{attribute addProperty BoxType "EP9224-0023-0016"}
{attribute addProperty Id "Temperature_WarningAT %I*BOOL811Temperature_ErrorAT %I*BOOL812Us_WarningAT %I*BOOL813Us_ErrorAT %I*BOOL814Up_WarningAT %I*BOOL815Up_ErrorAT %I*BOOL816Global_Error_BitAT %I*BOOL817Sum_Current_WarningAT %I*BOOL818Sum_Current_ErrorAT %I*BOOL819Reset_InputAT %I*BOOL8112TxPDO_StateAT %I*BOOL8115TxPDO_ToggleAT %I*BOOL8116Current_UsAT %I*INT16217Current_UpAT %I*INT16218Voltage_UsAT %I*INT16219Voltage_UpAT %I*INT16220TemperatureAT %I*INT16221"}
{attribute addProperty CRC "807253555"}
{attribute addProperty SizeInBites "176"}
{attribute addProperty SizeInBytes "22"}
TYPE DPO_Inputs_Device_301DB633 :
STRUCT
	{attribute addProperty Name "Temperature_Warning"}
	Temperature_Warning AT %I* : BOOL;
	{attribute addProperty Name "Temperature_Error"}
	Temperature_Error AT %I* : BOOL;
	{attribute addProperty Name "Us_Warning"}
	Us_Warning AT %I* : BOOL;
	{attribute addProperty Name "Us_Error"}
	Us_Error AT %I* : BOOL;
	{attribute addProperty Name "Up_Warning"}
	Up_Warning AT %I* : BOOL;
	{attribute addProperty Name "Up_Error"}
	Up_Error AT %I* : BOOL;
	{attribute addProperty Name "Global_Error_Bit"}
	Global_Error_Bit AT %I* : BOOL;
	{attribute addProperty Name "Sum_Current_Warning"}
	Sum_Current_Warning AT %I* : BOOL;
	{attribute addProperty Name "Sum_Current_Error"}
	Sum_Current_Error AT %I* : BOOL;
	{attribute addProperty Name "Reset_Input"}
	Reset_Input AT %I* : BOOL;
	{attribute addProperty Name "TxPDO_State"}
	TxPDO_State AT %I* : BOOL;
	{attribute addProperty Name "TxPDO_Toggle"}
	TxPDO_Toggle AT %I* : BOOL;
	{attribute addProperty Name "Current_Us"}
	Current_Us AT %I* : INT;
	{attribute addProperty Name "Current_Up"}
	Current_Up AT %I* : INT;
	{attribute addProperty Name "Voltage_Us"}
	Voltage_Us AT %I* : INT;
	{attribute addProperty Name "Voltage_Up"}
	Voltage_Up AT %I* : INT;
	{attribute addProperty Name "Temperature"}
	Temperature AT %I* : INT;
END_STRUCT
END_TYPE

(* stored: Version 1.2.0.0, ProductVersion 3.1.4024.9
   DUT DPO_Inputs_Device_301DB633: Id {c16f3127-d666-4e1f-8abe-9a41dfaa5710} *)
